FUNCTION_BLOCK server (* Tamplate for a simple Basic Function Block Type *)
  (* Standard: 61499-2 *)
  (* Version 0.0, 2018-06-06, 4DIAC-IDE, 4DIAC-Consortium *)
  (* Version 1.0, 2016-05-26, AZ, fortiss GmbH *)
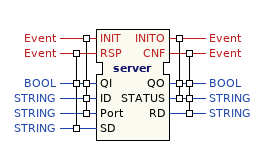
  EVENT_INPUT
    INIT WITH QI, ID, Port; (* Initialization Request *)
    RSP WITH QI, SD; (* Normal Execution Request *)
  END_EVENT
  EVENT_OUTPUT
    INITO WITH QO, STATUS; (* Initialization Confirm *)
    CNF WITH QO, STATUS, RD; (* Execution Confirmation *)
  END_EVENT
  VAR_INPUT
    QI : BOOL; (* Input event qualifier *)
    ID : STRING;
    Port : STRING;
    SD : STRING;
  END_VAR
  VAR_OUTPUT
    QO : BOOL; (* Output event qualifier *)
    STATUS : STRING;
    RD : STRING;
  END_VAR
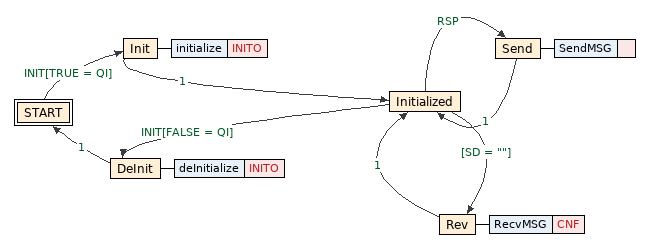
  EC_STATES
    START; (* Initial State *)
    Init : initialize -> INITO; (* Initialization *)
    Send : SendMSG; (* Normal execution *)
    Initialized;
    DeInit : deInitialize -> INITO;
    Rev : RecvMSG -> CNF;
  END_STATES
  EC_TRANSITIONS
    START TO Init := INIT[TRUE = QI];
    Init TO Initialized := 1;
    Initialized TO Send := RSP;
    DeInit TO START := 1;
    Initialized TO DeInit := INIT[FALSE = QI];
    Rev TO Initialized := 1;
    Send TO Initialized := 1;
    Initialized TO Rev := [SD = ""];
  END_TRANSITIONS
  ALGORITHM initialize IN ST: (* Initialization algorithm *)
QO := QI;
  END_ALGORITHM
  ALGORITHM deInitialize IN ST: (* Normally executed algorithm *)
QO := FALSE;
  END_ALGORITHM
  ALGORITHM SendMSG IN ST: (* new algorithm *)

  END_ALGORITHM
  ALGORITHM RecvMSG IN ST: (* new algorithm *)

  END_ALGORITHM
END_FUNCTION_BLOCK
